(* IEC 61131-3 sources: ATCMcontrol_Engineering/src/TargetBase/Libs/ATCM_CANopen, 8 files *)

(* ---- CANopen_BoardCmd.st ---- *)
(*[[
    UserURL= "ATCMfile:CANopen_BoardCmd.htm"
]]*)
FUNCTION CANopen_BoardCmd:DWORD

VAR_INPUT
   ExecMode:       INT;
END_VAR

VAR_OUTPUT
   ExecStatus:     DWORD;
END_VAR

VAR_INPUT
   Board:          INT;
   Command:        INT;
   CfgFileName:    STRING;
END_VAR

inline {STDLIB(CAN_BOARD_CMD)}

END_FUNCTION

(* ---- CANopen_GetEmcyInfo.st ---- *)
(*[[
    UserURL= "ATCMfile:CANopen_GetEmcyInfo.htm"
]]*)
FUNCTION CANopen_GetEmcyInfo:DWORD

VAR_INPUT
   ExecMode:       INT;
END_VAR

VAR_OUTPUT
   ExecStatus:     DWORD;
END_VAR

VAR_INPUT
   Board:          INT;
   NodeId:         INT;
   Timeout:        INT;
END_VAR

VAR_OUTPUT
   NodeStatus:     WORD;
   AddInfo:        WORD;
   ProfileNum:     INT;
   NodeState:      INT;
   ActualErr:      INT;
   EmcyLen:        INT;
   EmcyData: array[0..4] of CANopen_EmcyType;
END_VAR

inline { STDLIB(GET_EMCY_INFO) }

END_FUNCTION

(* ---- CANopen_GetEmcyNode.st ---- *)
(*[[
    UserURL= "ATCMfile:CANopen_GetEmcyNode.htm"
]]*)
FUNCTION CANopen_GetEmcyNode:DWORD

VAR_INPUT
   ExecMode:       INT;
END_VAR

VAR_OUTPUT
   ExecStatus:     DWORD;
END_VAR

VAR_INPUT
   Board:          INT;
END_VAR

VAR_IN_OUT
   NodeId:         INT;
END_VAR

inline {STDLIB(GET_EMCY_NODE)}

END_FUNCTION

(* ---- CANopen_GetStatus.st ---- *)
(*[[
    UserURL= "ATCMfile:CANopen_GetStatus.htm"
]]*)
FUNCTION CANopen_GetStatus:DWORD

VAR_INPUT
   ExecMode:       INT;
END_VAR

VAR_OUTPUT
   ExecStatus:     DWORD;
END_VAR

VAR_INPUT
   Board:          INT;
END_VAR

VAR_OUTPUT
   StatusData:     CANopen_StatusType;
END_VAR

inline { STDLIB(GET_STATUS) }

END_FUNCTION

(* ---- CANopen_NmtCmd.st ---- *)
(*[[
    UserURL= "ATCMfile:CANopen_NmtCmd.htm"
]]*)
FUNCTION CANopen_NmtCmd:DWORD

VAR_INPUT
   ExecMode:       INT;
END_VAR

VAR_OUTPUT
   ExecStatus:     DWORD;
END_VAR

VAR_INPUT
   Board:          INT;
   NodeId:         INT;
   Cmd:            INT;
   Timeout:        INT;
END_VAR

inline { STDLIB(NMT_CMD) }

END_FUNCTION

(* ---- CANopen_ReadSdoCmd.st ---- *)
(*[[
    UserURL= "ATCMfile:CANopen_ReadSdoCmd.htm"
]]*)
FUNCTION CANopen_ReadSdoCmd:DWORD

VAR_INPUT
   ExecMode:       INT;
END_VAR

VAR_OUTPUT
   ExecStatus:     DWORD;
END_VAR

VAR_INPUT
   Board:          INT;
   NodeId:         INT;
   Index:          WORD;
   subIndex:       INT;
   Timeout:        INT;
END_VAR

VAR_OUTPUT
 DataLength:       INT;
 Data:             ANY_ELEMENTARY;
END_VAR

overload DWORD(INT, DWORD, INT, INT, WORD, INT, INT, INT, BYTE)   inline { STDLIB(READ_SDO_CMD) }
overload DWORD(INT, DWORD, INT, INT, WORD, INT, INT, INT, INT)    inline { STDLIB(READ_SDO_CMD_W) }
overload DWORD(INT, DWORD, INT, INT, WORD, INT, INT, INT, WORD)   inline { STDLIB(READ_SDO_CMD_W) }
overload DWORD(INT, DWORD, INT, INT, WORD, INT, INT, INT, DINT)   inline { STDLIB(READ_SDO_CMD_DW) }
overload DWORD(INT, DWORD, INT, INT, WORD, INT, INT, INT, DWORD)  inline { STDLIB(READ_SDO_CMD_DW) }
overload DWORD(INT, DWORD, INT, INT, WORD, INT, INT, INT, STRING) inline { STDLIB(READ_SDO_CMD_S) }

END_FUNCTION

(* ---- CANopen_SyncCmd.st ---- *)
(*[[
    UserURL= "ATCMfile:CANopen_SyncCmd.htm"
]]*)
FUNCTION CANopen_SyncCmd:DWORD

VAR_INPUT
   ExecMode:       INT;
END_VAR

VAR_OUTPUT
   ExecStatus:     DWORD;
END_VAR

VAR_INPUT
   Board:          INT;
   Timeout:        INT;
END_VAR

inline {STDLIB(SYNC_CMD)}

END_FUNCTION

(* ---- CANopen_WriteSdoCmd.st ---- *)
(*[[
    UserURL= "ATCMfile:CANopen_WriteSdoCmd.htm"
]]*)
FUNCTION CANopen_WriteSdoCmd:DWORD

VAR_INPUT
   ExecMode:       INT;
END_VAR

VAR_OUTPUT
   ExecStatus:     DWORD;
END_VAR

VAR_INPUT
   Board:          INT;
   NodeId:         INT;
   Index:          WORD;
   subIndex:       INT;
   Timeout:        INT;
   DataLength:     INT;
END_VAR

VAR_IN_OUT
   Data:           ANY_ELEMENTARY;
END_VAR

overload DWORD(INT, DWORD, INT, INT, WORD, INT, INT, INT,  BYTE)   inline { STDLIB(WRITE_SDO_CMD) }
overload DWORD(INT, DWORD, INT, INT, WORD, INT, INT, INT,  INT)    inline { STDLIB(WRITE_SDO_CMD_W) }
overload DWORD(INT, DWORD, INT, INT, WORD, INT, INT, INT,  WORD)   inline { STDLIB(WRITE_SDO_CMD_W) }
overload DWORD(INT, DWORD, INT, INT, WORD, INT, INT, INT,  DINT)   inline { STDLIB(WRITE_SDO_CMD_DW) }
overload DWORD(INT, DWORD, INT, INT, WORD, INT, INT, INT,  DWORD)  inline { STDLIB(WRITE_SDO_CMD_DW) }
overload DWORD(INT, DWORD, INT, INT, WORD, INT, INT, INT,  STRING) inline { STDLIB(WRITE_SDO_CMD_S) }

END_FUNCTION
